(* CoDeSys 2.3 export: FB_LIMITOUTSIDEDOORCNTRL.EXP *)

(* POU new FB:s/FB_limitOutsideDoorCntrl, ST *)
FUNCTION_BLOCK FB_limitOutsideDoorCntrl
VAR_INPUT
	openInside				:BOOL;
	overSpeedLimit			:BOOL;
	doorInsideLimitOK		:BOOL;
END_VAR
VAR_OUTPUT
	ok							:BOOL;
END_VAR
VAR
END_VAR
IF overSpeedLimit THEN
	ok := FALSE;
ELSE IF openInside AND doorInsideLimitOK THEN
	ok:=TRUE;
END_IF;
END_FUNCTION_BLOCK
